{attribute addProperty BoxType "EL5101-0010-0016"}
{attribute addProperty Id "ENC_Status_compactAT %I*ENC_Status_compact_BE78AC8E4860ENC_Control_compactAT %Q*ENC_Control_compact_03701F333240WcStateAT %I*WcState_F855686C1620InfoDataAT %I*InfoData_BC63D37F80100"}
{attribute addProperty CRC "2727456817"}
{attribute addProperty SizeInBites "176"}
{attribute addProperty SizeInBytes "22"}
TYPE EL5101_AF3A94C8 :
STRUCT
	{attribute addProperty Name "ENC_Status_compact"}
	ENC_Status_compact : ENC_Status_compact_BE78AC8E;
	{attribute addProperty Name "ENC_Control_compact"}
	ENC_Control_compact : ENC_Control_compact_03701F33;
	{attribute addProperty Name "WcState"}
	WcState : WcState_F855686C;
	{attribute addProperty Name "InfoData"}
	InfoData : InfoData_BC63D37F;
END_STRUCT
END_TYPE

(* stored: Version 1.2.0.0, ProductVersion 3.1.4024.9
   DUT EL5101_AF3A94C8: Id {3da61043-dbb1-48ed-a905-2802d9f26042} *)
